RoboDK station: HAMK_Robotics_station_MG400_without_tool_example_program.rdk

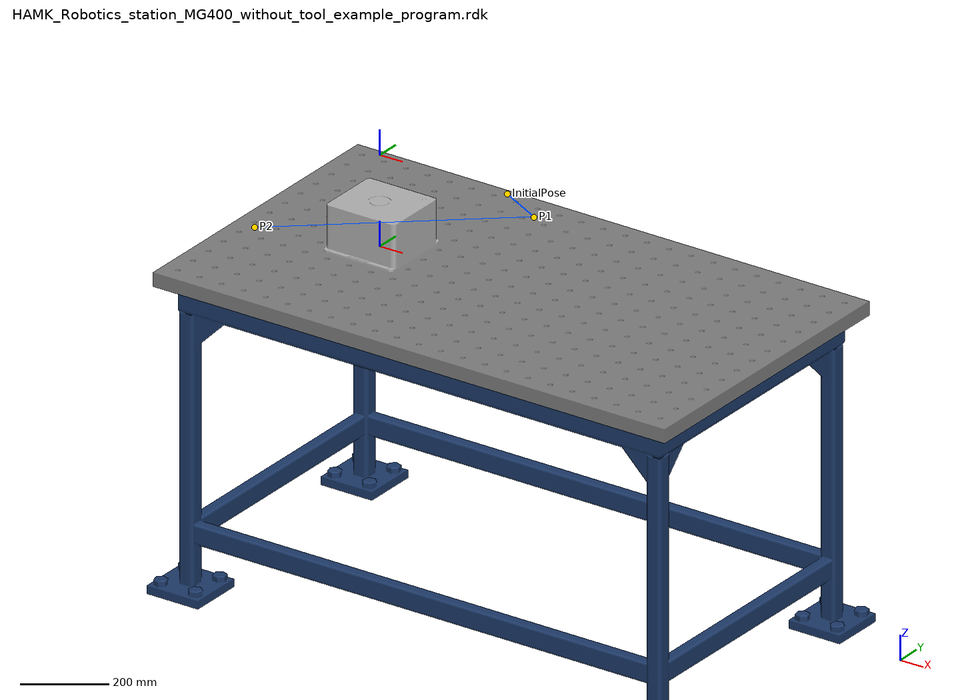
[picture v0: the station drawn from its stored meshes, robots at their saved joint values, targets as dots, program paths as lines]
Station HAMK_Robotics_station_MG400_without_tool_example_program (saved by RoboDK 5.8.0). Poses are relative to the parent item; angles as X-Y-Z fixed-axis rotations.
  - frame Dobot MG400 Base at (0, 0, 0) mm
    - robot Dobot MG400: 4 axes, payload 0.5 kg, reach 393.5 mm, repeatability 0.2 mm, weight 4 kg
        joint limits [-160, -25, -25, -360] to [160, 85, 105, 360]; home [0, 0, 0, 0]; saved at [0, 32.158, 32.645, 0]
      - tool MG400_End_Flange, TCP at (0, 0, -13) mm, size 39.8 x 39.8 x 14 mm
    - frame World at (0, 0, 0) mm
      - object Table 1400x800x800mm at (0, 0, 0) mm, size 1420 x 820 x 800 mm, geometry from Table-1400x800x800mm.sld
        - object HAMK logo at (360, 380, -115) mm, rotated rx 90 ry 0 rz 180 deg, size 301.4 x 100.9 x 9.4 mm, geometry from Fantastic Duup(2).stl
        - object white background at (360, 385.5, -110) mm, rotated rx 90 ry 0 rz 0 deg, size 480 x 184.8 x 2.4 mm, geometry from Fantastic Duup(3).stl
  - frame ReferenceFrameTCP at (0, 0, 227.75) mm
    - target InitialPose (Cartesian target) at (350, 0, 0) mm; joints [0, 32.158, 32.645, 0] of Dobot MG400
    - target P1 (Cartesian target) at (290, 190, -150) mm; joints [33.232, 69.088, 65.084, 33.232] of Dobot MG400
    - target P2 (Cartesian target) at (-110, -330, -80) mm; joints [-108.435, 49.53, 53.04, -108.435] of Dobot MG400
  - program Prog1 (6 instructions, listed below)
  - notes Note 1: <!DOCTYPE HTML PUBLIC "-//W3C//DTD HTML 4.0//EN" "http://www.w3.org/TR/REC-html40/strict.dtd">
<html><head><meta name="qrichtext" content="1" /><style type="text/css">
p, li { white-space: pre-wrap; }
</style></head><body style=" font-family:'MS Shell Dlg 2'; font-size:7.8pt; font-weight:400; font-style:normal;">
<p style=" margin-top:0px; margin-bottom:0px; margin-left:0px; margin-right:0px; -qt-block-indent:0; text-indent:0px;">In this station, a dummy tool (only the flange downloaded from https://uptimefab.com/2022/02/07/dobot-mg400/) is added to consider the 13mm of the tool shaft. Then, we use the coordinates of the TCP, that is, of the tip of the tool shaft.</p>
<p style=" margin-top:0px; margin-bottom:0px; margin-left:0px; margin-right:0px; -qt-block-indent:0; text-indent:0px;">Without any tool, the coordinates are refered to the robot flange.</p>
<p style=" margin-top:0px; margin-bottom:0px; margin-left:0px; margin-right:0px; -qt-block-indent:0; text-indent:0px;">Fernando S. Pacheco</p>
<p style=" margin-top:0px; margin-bottom:0px; margin-left:0px; margin-right:0px; -qt-block-indent:0; text-indent:0px;">September 2024</p>
<p style="-qt-paragraph-type:empty; margin-top:0px; margin-bottom:0px; margin-left:0px; margin-right:0px; -qt-block-indent:0; text-indent:0px;"><br /></p></body></html>
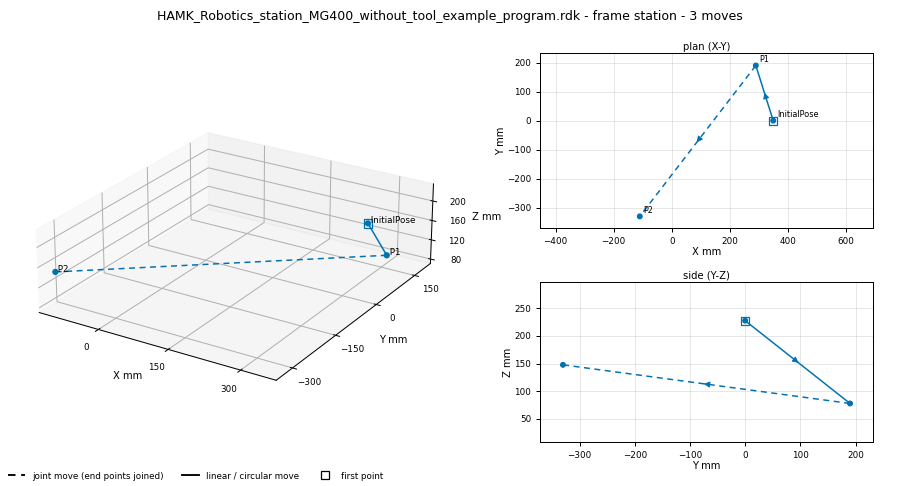
[picture p0: tool path of HAMK_Robotics_station_MG400_without_tool_example_program.rdk in frame station, 3 of 3 moves have a stored position in this frame; points joined in program order, loops and branches not executed]

--- program Prog1 (robot Dobot MG400) ---
  This program should have exactly the same result as one with DobotStudio Blockly.
  Set Ref.: ReferenceFrameTCP
  Set Tool: MG400_End_Flange
  MoveJ (InitialPose)
  MoveL (P1)
  MoveJ (P2)
